{attribute 'hide_all_locals'}
FUNCTION_BLOCK PUBLIC ABSTRACT FB_Employee IMPLEMENTS I_Employee
VAR_INPUT
END_VAR
VAR_OUTPUT
END_VAR
VAR
	nPersonnelNumberBacking :	UINT;
	sFirstNameBacking		:	STRING;
	sLastNameBacking		:	STRING;
END_VAR

METHOD PUBLIC GetFullName : STRING
VAR_INPUT
END_VAR
GetFullName := CONCAT(CONCAT(CONCAT(CONCAT(TO_STRING(nPersonnelNumber), ': '), sFirstName), ' '), sLastName);
END_METHOD

METHOD PUBLIC ABSTRACT GetMonthlySalary : LREAL
VAR_INPUT
END_VAR
END_METHOD

{attribute 'monitoring' := 'variable'}
PROPERTY PUBLIC nPersonnelNumber : UINT
GET
nPersonnelNumber := nPersonnelNumberBacking;
END_GET
SET
nPersonnelNumberBacking := nPersonnelNumber;
END_SET
END_PROPERTY

{attribute 'monitoring' := 'variable'}
PROPERTY PUBLIC sFirstName : STRING
GET
sFirstName := sFirstNameBacking;
END_GET
SET
sFirstNameBacking := sFirstName;
END_SET
END_PROPERTY

{attribute 'monitoring' := 'variable'}
PROPERTY PUBLIC sLastName : STRING
GET
sLastName := sLastNameBacking;
END_GET
SET
sLastNameBacking := sLastName;
END_SET
END_PROPERTY

END_FUNCTION_BLOCK

(* stored: Version 1.1.0.1, ProductVersion 3.1.4024.4
   POU FB_Employee: Id {2cc7defd-3e09-4270-815e-92d7c2b9e2ed}, SpecialFunc None
   Method GetFullName: Id {a38adcfd-bdb3-4984-8ca9-9695a28e2a21}
   Method GetMonthlySalary: Id {c2c84659-4bba-4b37-8367-127abc5f70e0}
   Property nPersonnelNumber: Id {7eca07d9-ded1-4ef4-8f6f-f1a39ae6d112}
   Get Get: Id {1f8d65b6-a3a5-4864-9561-584b659cde32}
   Set Set: Id {c77b21f5-0e83-47d0-b8c9-df3b029cf132}
   Property sFirstName: Id {b4a086ca-225d-476d-8efa-e89be1aaab40}
   Get Get: Id {8cf9f14d-a12b-4d65-88aa-1965682651c1}
   Set Set: Id {c5459749-aad0-45e3-9435-cf39ee597117}
   Property sLastName: Id {2b72463c-3390-4d6c-b808-2f94b0f06cc4}
   Get Get: Id {0e328a25-766a-4e02-9bde-edeb61c794dc}
   Set Set: Id {367abf85-df4b-4da9-9b37-3e0dbf5ac2c6} *)
